FUNCTION_BLOCK "Block_1"
{ S7_Optimized_Access := 'TRUE' }
VERSION : 0.1
   VAR_INPUT
      hej : Bool;
   END_VAR


BEGIN
END_FUNCTION_BLOCK

